TYPE ST_IotData_credits :
STRUCT
	TotalCredits 		: DINT := 100;
	RemainingCredits	: DINT;
	UsedCredits			: DINT;
END_STRUCT
END_TYPE

(* stored: Version 1.1.0.1, ProductVersion 3.1.4026.18
   DUT ST_IotData_credits: Id {84eae8b9-871b-4556-8a8e-03a11a78039d} *)
